FUNCTION_BLOCK FB_Mx_FP_Reset			// FB zum erkennen einer steigender Flanke
VAR_INPUT
	Ix_Reset: BOOL;						// Abzufragendes Signal
END_VAR
VAR_OUTPUT
END_VAR
VAR
	Mx_lmp_Reset: BOOL;					// Ausgang für 1 Zyklus aktiv wenn negativepositive Flanke erkannt
	last_CLK: BOOL;						// Zwischenspeicher des letzten Zustandes des Eingangssignal
END_VAR

Mx_lmp_Reset:= Ix_Reset AND NOT last_CLK;
last_CLK:= Ix_Reset;

END_FUNCTION_BLOCK

(* stored: Version 1.1.0.1
   POU FB_Mx_FP_Reset: Id {9c891d4c-1c8e-487b-a4f2-8c0a646bd387}, SpecialFunc None *)
